{attribute 'strict'}
{attribute 'qualified_only'}
TYPE E_LineMachineCommand :
(
	eAbort	  				:= 10,
	eStop	  				:= 20,
	eRun	  				:= 30,
	eReset	  				:= 40,
	eRestart 				:= 50,
	ePause					:= 60
);
END_TYPE

(* stored: Version 1.1.0.1, ProductVersion 3.1.4022.12
   DUT E_LineMachineCommand: Id {ed4e1a30-40dc-4b59-9130-9965c0e0ecde} *)
